FUNCTION_BLOCK FB_ProBoxElement2Motor EXTENDS FB_ProBoxElementBase
(**************************************************************************************
 * 	Application		:	BoxControl Framework
 *	Revision		:	$Revision:  $
 *	Revision date	:	$Date:  $
 *	Last changed by	:	$Author:  $
 *	URL				:	$URL: $
 *
 *	Purpose			:	ProBox element with 2 axis and 2 motor HW outputs (drive 1-2 / 3-4).
 *
 * ------------------------------------------------------------------------------------
 *	Copyright Swisslog [IP AG], Switzerland. All rights reserved.
 * 
 * ------------------------------------------------------------------------------------
 *	
 * 	Revision History: 
 *
 * 	VERSION			DATE			INITIALS			DESCRIPTION
 *	
 *
 **************************************************************************************)
VAR_INPUT
	Config					: ST_CFG_ProBoxElementMotor; // Configuration 
	HW_Inputs				: ST_HW_InputsProBoxElementMotor; // HW-Inputs 
END_VAR

VAR_OUTPUT
	HW_Outputs				: ST_HW_OutputsProBoxElement2Motor; // HW-Outputs 
END_VAR

VAR PERSISTENT
	Settings				: ST_CFG_ProBoxElementMotor; // Settings - activated configuration 
END_VAR


(**************************************************************************************************************
   Input mapping
***************************************************************************************************************)
A_InputMapping();


(**************************************************************************************************************
   Initialization
***************************************************************************************************************)
A_Init();


(**************************************************************************************************************
   State control
***************************************************************************************************************)
A_StateControl();


(**************************************************************************************************************
   Error handler
***************************************************************************************************************)
M_MonitorElementErrors();


(**************************************************************************************************************
   Manual control
***************************************************************************************************************)
A_ManualControl();


(**************************************************************************************************************
   Handle element functions
***************************************************************************************************************)
A_HandleFunctions();



(**********************************************************************************************************
   Drive control
***********************************************************************************************************)
A_DriveControl();



(**************************************************************************************************************
   Interface handler out
***************************************************************************************************************)
M_ITC_ProcessOut();


(**************************************************************************************************************
   Output mapping
***************************************************************************************************************)
A_OutputMapping();

ACTION A_Init:
(**************************************************************************************
 * 	NAME		A_Init
 * 	FUNCTION	Initialize element
 **************************************************************************************)
 
 IF NOT ElementData.Init AND NOT ElementData.InitRunning THEN
	 // Load function specific configuration to settings
	Settings := Config;
	SUPER^.BaseSettings.BrakeTime := Settings.BrakeTime;
	SUPER^.BaseSettings.ElementSpeed := Settings.ElementSpeed;
 END_IF
 
SUPER^.A_Init();
END_ACTION

ACTION A_InputMapping:
(**************************************************************************************
 * 	NAME		A_InputMapping
 * 	FUNCTION	Input mapping
 **************************************************************************************)
 
 
(**************************************************************************************
   Map HW Inputs
***************************************************************************************)
Inputs.MotorUnitOK := HW_Inputs.MotorUnitOK;
Super^.A_InputMapping();
END_ACTION

ACTION A_OutputMapping:
(**************************************************************************************
 * 	NAME		A_OutputMapping
 * 	FUNCTION	Handles element specific outpus
 **************************************************************************************)

(**************************************************************************************
   Map HW Outputs
***************************************************************************************)
HW_Outputs.Drive_Run_12		:= fbProBoxMotorControl_12.Forward;
HW_Outputs.Drive_Run_21		:= fbProBoxMotorControl_12.Reverse;
HW_Outputs.Drive_Creep_12	:= fbProBoxMotorControl_12.CreepSpeed;
HW_Outputs.Drive_Low_12		:= fbProBoxMotorControl_12.LowSpeed;
HW_Outputs.MotorBrake_12	:= fbProBoxMotorControl_12.BrakeRelease;

HW_Outputs.Drive_Run_34		:= fbProBoxMotorControl_34.Forward;
HW_Outputs.Drive_Run_43		:= fbProBoxMotorControl_34.Reverse;
HW_Outputs.Drive_Creep_34	:= fbProBoxMotorControl_34.CreepSpeed;
HW_Outputs.Drive_Low_34		:= fbProBoxMotorControl_34.LowSpeed;
HW_Outputs.MotorBrake_34	:= fbProBoxMotorControl_34.BrakeRelease;
 
(**************************************************************************************
   Map element interface
***************************************************************************************)

// interface axis 1-2
SUPER^.A_OutputMapping();
END_ACTION

END_FUNCTION_BLOCK

(* stored: Version 1.1.0.1, ProductVersion 3.1.4024.9
   POU FB_ProBoxElement2Motor: Id {a45382ee-1b1f-422f-87e8-f05701e775fc}, SpecialFunc None
   Action A_Init: Id {0905c26f-ada7-4d29-aa05-19de42a7e78d}
   Action A_InputMapping: Id {fa01f38a-9c49-45e0-bcc3-f318ca71a8c7}
   Action A_OutputMapping: Id {ba5ac88a-ca62-48ba-8069-7d572c284ff1} *)
